// TIA Portal V16 program export: 1 tag tables, 0 data types, 0 data blocks, 1 code blocks (in call order from the OBs), 0 instance data blocks

VAR_GLOBAL   // PLC tag table "TwoWay_Switch(XOR)"
   Stop AT %I0.0 : Bool;
   Switch_1 AT %I0.1 : Bool;
   Switch_2 AT %I0.2 : Bool;
   Lamba AT %Q0.0 : Bool;
END_VAR

ORGANIZATION_BLOCK "TwoWay_Switch(XOR)"   // OB1, LAD, ProgramCycle
TITLE = "Main Program Sweep (Cycle)"
{ S7_Optimized_Access := 'TRUE' }
VERSION : 0.1
// stored: AutoNumber true, IsIECCheckEnabled false, SetENOAutomatically false
   VAR_INPUT
      Initial_Call : Bool;   // Initial call of this OB
      Remanence : Bool;   // =True, if remanent data are available
   END_VAR
BEGIN

REGION Network 1
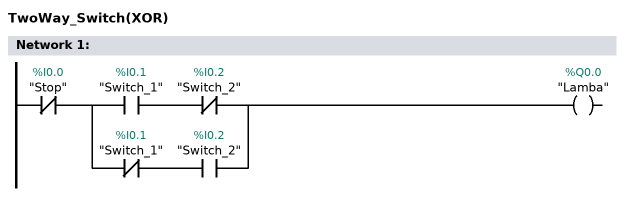
   RUNG wire#powerrail
      I_Contact( "Stop" )
      wire#w1
      Contact( "Switch_1" )
      I_Contact( "Switch_2" )
      wire#w2
      Coil( "Lamba" )
   END_RUNG
   RUNG wire#w1
      I_Contact( "Switch_1" )
      Contact( "Switch_2" )
   END_RUNG wire#w2
   // the same network as SCL:
   "Lamba" := NOT "Stop" AND (("Switch_1" AND NOT "Switch_2") OR (NOT "Switch_1" AND "Switch_2"));
END_REGION
END_ORGANIZATION_BLOCK
